{attribute 'GeneratedUsingTerminal: BK1250-0000-0019'}
{attribute addProperty BoxType "BK1250-0000-0019"}
{attribute addProperty Id "A_0001_KL_6211_ASI_Master_Parameter_Interface_and_6_Byte_11_ASI_Slaves_PowerKL6211_60136EA10A_0002_KL_6211_ASI_Master_Parameter_Interface_and_6_Byte_11_ASI_Slaves_PowerKL_9AE543B60A_0005_KL_6211_ASI_Master_Parameter_Interface_and_16_Byte_31_ASI_Slaves_PowerKL_FC0201B80A_0006_KL_6211_ASI_Master_Parameter_Interface_and_16_Byte_31_ASI_Slaves_PowerKL_498D88630A_0009_KL_6211_ASI_Master_Parameter_Interface_and_32_Byte_62_ASI_Slaves_PowerKL_713416910A_0010_KL_6211_ASI_Master_Parameter_Interface_and_32_Byte_62_ASI_Slaves_PowerKL_2B11657C0A_0012_KL_6224_IO_Link_Master_Parameter_Interface_and_6_Byte_Process_DataKL6224_C0F107BD0A_0013_KL_6224_IO_Link_Master_Parameter_Interface_and_18_Byte_Process_DataKL_FC1E33930A_0014_KL_6224_IO_Link_Master_Parameter_Interface_and_30_Byte_Process_DataKL_C51B1CB00A_0015_KL_6224_IO_Link_Master_Parameter_Interface_and_42_Byte_Process_DataKL_7EC2CD640A_0016_KL_6301_EIB_24_BYTE_InterfaceKL_3829421A0A_0017_KL_6401_LON_36_BYTE_InterfaceKL_9116C2C10A_0018_KM_6551_IEEE802_15_4_12_Byte_InterfaceKL6551_528AE3980A_0019_KL_6581_EnOcean_12_BYTE_InterfaceKL_3325E5830A_0020_KM_6663_Ethernet_Changeover_SwitchKL_DCA756120A_0021_KL_6771_MP_BUS_Master_12_Byte_InterfaceKL_528AE3980A_0022_KL_6781_M_Bus_Interface_22_Byte_xKL6781_BE595CA20A_0023_KL_6811_DALI_Master_with_Power_SupplierKL6811_6148C9040A_0024_KL_6821_DALI_2_Multi_Master_with_Power_SupplierKL6821_F77C82D20A_0025_KL_6831_SMI_LoVo_Interface_22_Byte_xKL6831_BE595CA20A_0026_KL_6841_SMI_AC_Interface_22_Byte_xKL6841_BE595CA20A_0027_KL_6904_Safety_Logic_7_TwinSAFE_ConnectionsKL6904_B938D6120A_0028_KL_6904_Safety_Logic_15_TwinSAFE_ConnectionsKL_921B772D0A_0029_KL_8001_Powerterminal_1ChKL_779990DF0A_0030_KL_8001_Powerterminal_3_ChKL8001_7761653A0A_0031_KL_8519_16_digital_InputKL8519_8C34650F0A_0032_KL_8524_2x4_digital_OutputKL8524_A4B9216E0A_0033_KL_8528_8_digital_OutputKL8528_73A97EC10A_0034_KL_8548_8_Ch_ana_Output_0_10VKL8548_234517280A_0035_KL_8610_1_Ch_Adapter_KL8601KL8610_C571D0680A_0036_KL_8610_2_Ch_Adapter_KL8601KL_5A83E84C0A_0037_KL_8610_3_Ch_Adapter_KL8601KL_BF4AA06C0A_0038_KL_8610_4_Ch_Adapter_KL8601KL_7485E9250A_0039_KL_8610_5_Ch_Adapter_KL8601KL_372C6BEC0A_0040_KL_8610_6_Ch_Adapter_KL8601KL_2E5CD6C80A_0041_KL_8610_7_Ch_Adapter_KL8601KL_68BDE1E90A_0042_KL_8610_8_Ch_Adapter_KL8601KL_84AAE8B60A_0050_KL_9110_Power_Supplier_with_LED_and_Diag_24VKL9110_8BEE55F20A_0052_KL_9160_Power_Supplier_with_LED_and_Diag_230VKL9160_8BEE55F20A_0064_KL_9191_Dig_I_OKL9191_962A24DF0A_0067_KL_9210_Power_Supplier_with_Fuse_LED_and_Diag_24VKL9210_8BEE55F20A_0069_KL_9260_Power_Supplier_with_Fuse_LED_and_Diag_230VKL9260_8BEE55F20A_0078_KL_9505_0010_Power_Supplier_5V_0_5A_DiagKL_E4BD2B380A_0080_KL_9508_0010_Power_Supplier_8V_0_5A_DiagKL_E4BD2B380A_0082_KL_9510_0010_Power_Supplier_10V_0_5A_DiagKL_E4BD2B380A_0084_KL_9512_0010_Power_Supplier_12V_0_5A_DiagKL_E4BD2B380A_0086_KL_9515_0010_Power_Supplier_15V_0_5A_DiagKL_E4BD2B380A_0087_KL_9528_Power_Supplier_AS_i_2AKL9528_8C9846030A_0092_KLWORD_1_In_and_1_Output_WordKL9999_7A10A7F60"}
{attribute addProperty CRC "3472310613"}
{attribute addProperty Size "0"}
TYPE TcTerminals210_2BK1250_CEF74155 EXTENDS BK1250_AEEC0900 :
STRUCT
	{attribute addProperty Name "A_0001_KL_6211_ASI_Master_Parameter_Interface_and_6_Byte_11_ASI_Slaves_Power"}
	A_0001_KL_6211_ASI_Master_Parameter_Interface_and_6_Byte_11_ASI_Slaves_Power : KL6211_60136EA1;
	{attribute addProperty Name "A_0002_KL_6211_ASI_Master_Parameter_Interface_and_6_Byte_11_ASI_Slaves_Power"}
	A_0002_KL_6211_ASI_Master_Parameter_Interface_and_6_Byte_11_ASI_Slaves_Power : KL_9AE543B6;
	{attribute addProperty Name "A_0005_KL_6211_ASI_Master_Parameter_Interface_and_16_Byte_31_ASI_Slaves_Power"}
	A_0005_KL_6211_ASI_Master_Parameter_Interface_and_16_Byte_31_ASI_Slaves_Power : KL_FC0201B8;
	{attribute addProperty Name "A_0006_KL_6211_ASI_Master_Parameter_Interface_and_16_Byte_31_ASI_Slaves_Power"}
	A_0006_KL_6211_ASI_Master_Parameter_Interface_and_16_Byte_31_ASI_Slaves_Power : KL_498D8863;
	{attribute addProperty Name "A_0009_KL_6211_ASI_Master_Parameter_Interface_and_32_Byte_62_ASI_Slaves_Power"}
	A_0009_KL_6211_ASI_Master_Parameter_Interface_and_32_Byte_62_ASI_Slaves_Power : KL_71341691;
	{attribute addProperty Name "A_0010_KL_6211_ASI_Master_Parameter_Interface_and_32_Byte_62_ASI_Slaves_Power"}
	A_0010_KL_6211_ASI_Master_Parameter_Interface_and_32_Byte_62_ASI_Slaves_Power : KL_2B11657C;
	{attribute addProperty Name "A_0012_KL_6224_IO_Link_Master_Parameter_Interface_and_6_Byte_Process_Data"}
	A_0012_KL_6224_IO_Link_Master_Parameter_Interface_and_6_Byte_Process_Data : KL6224_C0F107BD;
	{attribute addProperty Name "A_0013_KL_6224_IO_Link_Master_Parameter_Interface_and_18_Byte_Process_Data"}
	A_0013_KL_6224_IO_Link_Master_Parameter_Interface_and_18_Byte_Process_Data : KL_FC1E3393;
	{attribute addProperty Name "A_0014_KL_6224_IO_Link_Master_Parameter_Interface_and_30_Byte_Process_Data"}
	A_0014_KL_6224_IO_Link_Master_Parameter_Interface_and_30_Byte_Process_Data : KL_C51B1CB0;
	{attribute addProperty Name "A_0015_KL_6224_IO_Link_Master_Parameter_Interface_and_42_Byte_Process_Data"}
	A_0015_KL_6224_IO_Link_Master_Parameter_Interface_and_42_Byte_Process_Data : KL_7EC2CD64;
	{attribute addProperty Name "A_0016_KL_6301_EIB_24_BYTE_Interface"}
	A_0016_KL_6301_EIB_24_BYTE_Interface : KL_3829421A;
	{attribute addProperty Name "A_0017_KL_6401_LON_36_BYTE_Interface"}
	A_0017_KL_6401_LON_36_BYTE_Interface : KL_9116C2C1;
	{attribute addProperty Name "A_0018_KM_6551_IEEE802_15_4_12_Byte_Interface"}
	A_0018_KM_6551_IEEE802_15_4_12_Byte_Interface : KL6551_528AE398;
	{attribute addProperty Name "A_0019_KL_6581_EnOcean_12_BYTE_Interface"}
	A_0019_KL_6581_EnOcean_12_BYTE_Interface : KL_3325E583;
	{attribute addProperty Name "A_0020_KM_6663_Ethernet_Changeover_Switch"}
	A_0020_KM_6663_Ethernet_Changeover_Switch : KL_DCA75612;
	{attribute addProperty Name "A_0021_KL_6771_MP_BUS_Master_12_Byte_Interface"}
	A_0021_KL_6771_MP_BUS_Master_12_Byte_Interface : KL_528AE398;
	{attribute addProperty Name "A_0022_KL_6781_M_Bus_Interface_22_Byte_x"}
	A_0022_KL_6781_M_Bus_Interface_22_Byte_x : KL6781_BE595CA2;
	{attribute addProperty Name "A_0023_KL_6811_DALI_Master_with_Power_Supplier"}
	A_0023_KL_6811_DALI_Master_with_Power_Supplier : KL6811_6148C904;
	{attribute addProperty Name "A_0024_KL_6821_DALI_2_Multi_Master_with_Power_Supplier"}
	A_0024_KL_6821_DALI_2_Multi_Master_with_Power_Supplier : KL6821_F77C82D2;
	{attribute addProperty Name "A_0025_KL_6831_SMI_LoVo_Interface_22_Byte_x"}
	A_0025_KL_6831_SMI_LoVo_Interface_22_Byte_x : KL6831_BE595CA2;
	{attribute addProperty Name "A_0026_KL_6841_SMI_AC_Interface_22_Byte_x"}
	A_0026_KL_6841_SMI_AC_Interface_22_Byte_x : KL6841_BE595CA2;
	{attribute addProperty Name "A_0027_KL_6904_Safety_Logic_7_TwinSAFE_Connections"}
	A_0027_KL_6904_Safety_Logic_7_TwinSAFE_Connections : KL6904_B938D612;
	{attribute addProperty Name "A_0028_KL_6904_Safety_Logic_15_TwinSAFE_Connections"}
	A_0028_KL_6904_Safety_Logic_15_TwinSAFE_Connections : KL_921B772D;
	{attribute addProperty Name "A_0029_KL_8001_Powerterminal_1Ch"}
	A_0029_KL_8001_Powerterminal_1Ch : KL_779990DF;
	{attribute addProperty Name "A_0030_KL_8001_Powerterminal_3_Ch"}
	A_0030_KL_8001_Powerterminal_3_Ch : KL8001_7761653A;
	{attribute addProperty Name "A_0031_KL_8519_16_digital_Input"}
	A_0031_KL_8519_16_digital_Input : KL8519_8C34650F;
	{attribute addProperty Name "A_0032_KL_8524_2x4_digital_Output"}
	A_0032_KL_8524_2x4_digital_Output : KL8524_A4B9216E;
	{attribute addProperty Name "A_0033_KL_8528_8_digital_Output"}
	A_0033_KL_8528_8_digital_Output : KL8528_73A97EC1;
	{attribute addProperty Name "A_0034_KL_8548_8_Ch_ana_Output_0_10V"}
	A_0034_KL_8548_8_Ch_ana_Output_0_10V : KL8548_23451728;
	{attribute addProperty Name "A_0035_KL_8610_1_Ch_Adapter_KL8601"}
	A_0035_KL_8610_1_Ch_Adapter_KL8601 : KL8610_C571D068;
	{attribute addProperty Name "A_0036_KL_8610_2_Ch_Adapter_KL8601"}
	A_0036_KL_8610_2_Ch_Adapter_KL8601 : KL_5A83E84C;
	{attribute addProperty Name "A_0037_KL_8610_3_Ch_Adapter_KL8601"}
	A_0037_KL_8610_3_Ch_Adapter_KL8601 : KL_BF4AA06C;
	{attribute addProperty Name "A_0038_KL_8610_4_Ch_Adapter_KL8601"}
	A_0038_KL_8610_4_Ch_Adapter_KL8601 : KL_7485E925;
	{attribute addProperty Name "A_0039_KL_8610_5_Ch_Adapter_KL8601"}
	A_0039_KL_8610_5_Ch_Adapter_KL8601 : KL_372C6BEC;
	{attribute addProperty Name "A_0040_KL_8610_6_Ch_Adapter_KL8601"}
	A_0040_KL_8610_6_Ch_Adapter_KL8601 : KL_2E5CD6C8;
	{attribute addProperty Name "A_0041_KL_8610_7_Ch_Adapter_KL8601"}
	A_0041_KL_8610_7_Ch_Adapter_KL8601 : KL_68BDE1E9;
	{attribute addProperty Name "A_0042_KL_8610_8_Ch_Adapter_KL8601"}
	A_0042_KL_8610_8_Ch_Adapter_KL8601 : KL_84AAE8B6;
	{attribute addProperty Name "A_0050_KL_9110_Power_Supplier_with_LED_and_Diag_24V"}
	A_0050_KL_9110_Power_Supplier_with_LED_and_Diag_24V : KL9110_8BEE55F2;
	{attribute addProperty Name "A_0052_KL_9160_Power_Supplier_with_LED_and_Diag_230V"}
	A_0052_KL_9160_Power_Supplier_with_LED_and_Diag_230V : KL9160_8BEE55F2;
	{attribute addProperty Name "A_0064_KL_9191_Dig_I_O"}
	A_0064_KL_9191_Dig_I_O : KL9191_962A24DF;
	{attribute addProperty Name "A_0067_KL_9210_Power_Supplier_with_Fuse_LED_and_Diag_24V"}
	A_0067_KL_9210_Power_Supplier_with_Fuse_LED_and_Diag_24V : KL9210_8BEE55F2;
	{attribute addProperty Name "A_0069_KL_9260_Power_Supplier_with_Fuse_LED_and_Diag_230V"}
	A_0069_KL_9260_Power_Supplier_with_Fuse_LED_and_Diag_230V : KL9260_8BEE55F2;
	{attribute addProperty Name "A_0078_KL_9505_0010_Power_Supplier_5V_0_5A_Diag"}
	A_0078_KL_9505_0010_Power_Supplier_5V_0_5A_Diag : KL_E4BD2B38;
	{attribute addProperty Name "A_0080_KL_9508_0010_Power_Supplier_8V_0_5A_Diag"}
	A_0080_KL_9508_0010_Power_Supplier_8V_0_5A_Diag : KL_E4BD2B38;
	{attribute addProperty Name "A_0082_KL_9510_0010_Power_Supplier_10V_0_5A_Diag"}
	A_0082_KL_9510_0010_Power_Supplier_10V_0_5A_Diag : KL_E4BD2B38;
	{attribute addProperty Name "A_0084_KL_9512_0010_Power_Supplier_12V_0_5A_Diag"}
	A_0084_KL_9512_0010_Power_Supplier_12V_0_5A_Diag : KL_E4BD2B38;
	{attribute addProperty Name "A_0086_KL_9515_0010_Power_Supplier_15V_0_5A_Diag"}
	A_0086_KL_9515_0010_Power_Supplier_15V_0_5A_Diag : KL_E4BD2B38;
	{attribute addProperty Name "A_0087_KL_9528_Power_Supplier_AS_i_2A"}
	A_0087_KL_9528_Power_Supplier_AS_i_2A : KL9528_8C984603;
	{attribute addProperty Name "A_0092_KLWORD_1_In_and_1_Output_Word"}
	A_0092_KLWORD_1_In_and_1_Output_Word : KL9999_7A10A7F6;
END_STRUCT
END_TYPE

(* stored: Version 1.2.0.0, ProductVersion 3.1.4024.9
   DUT TcTerminals210_2BK1250_CEF74155: Id {171fcb36-db62-4f12-a31a-1d8dbda81f13} *)
